(* Logix 5000 project; controller SS1 Emulate 5570 rev 36.11; software revision 36.00 *)

TASK MainTask (continuous, watchdog 500 ms) : MainProgram

MODULES
   Local : Emulate 5570 (ICP 2, rev 36.11)
       : 1756-IB16 (ICP 3, rev 3.1, Input RPI 20 ms)
       : 1756-OB16D (ICP 4, rev 3.1, Output RPI 20 ms)
END_MODULES

VAR_GLOBAL   (* controller tags *)
   MOTOR : ALIAS FOR Local:4:O.Data.2;   // Motor Control
   PL1_OFF : ALIAS FOR Local:4:O.Data.0;   // Pilot Light 1 OFF (Red)
   PL2_ON : ALIAS FOR Local:4:O.Data.1;   // Pilot Light 1 ON (Green)
   START : ALIAS FOR Local:3:I.Data.1;   // Pushbutton Momentary N.O.
   STOP : ALIAS FOR Local:3:I.Data.0;   // Pushbutton Momentary N.C.
END_VAR

PROGRAM MainProgram   (* main routine TextRoutine *)

ROUTINE TextRoutine   (* structured text *)
   //START-STOP pushbuttons to turn On MOTOR
   MOTOR := STOP AND (START OR MOTOR );
   
   //Indicators status based on MOTOR On or Off
   PL1_OFF:= NOT MOTOR ;
   PL2_ON[:=] MOTOR;
   
END_ROUTINE
END_PROGRAM
